# EPICS autosave request: motorApp/Db/XPSPositionCompare_settings.req
$(P)$(R)PositionCompareMode
$(p)$(r)pOSITIONcompareMinPosition
$(P)$(R)PositionCompareMaxPosition
$(P)$(R)PositionCompareStepSize
$(P)$(R)PositionComparePulseWidth
$(P)$(R)PositionCompareSettlingTime
